SYSTEM MSFUji
  (* Version 1.0, 2021-07-06, HP *)
  APPLICATION MSFFApp
    FBS
      E_CYCLE : E_CYCLE(DT := T#10ms);
      Stage3 : Stage3(DT := 0.01);
      Stage4 : Stage4(DT := 0.01);
      Stage5 : Stage5(DT := 0.01);
      Stage6 : Stage6(DT := 0.01);
      Stage7 : Stage7(DT := 0.01);
      Stage8 : Stage8(DT := 0.01);
      Stage9 : Stage9(DT := 0.01);
      Stage10 : Stage10(DT := 0.01);
      Stage11 : Stage11(DT := 0.01);
      Stage12 : Stage12(DT := 0.01);
      Stage13 : Stage13(DT := 0.01);
      Stage14 : Stage14(DT := 0.01);
      Stage15 : Stage15(DT := 0.01);
      Stage16 : Stage16(DT := 0.01);
      Stage17 : Stage17(DT := 0.01);
      Stage18 : Stage18(DT := 0.01);
      Stage19 : Stage19(DT := 0.01);
      Stage20 : Stage20(WFset := 143.81, DT := 0.01);
      Stage21 : Stage21(DT := 0.01);
      Stagesss22 : Stagesss22(DT := 0.01);
      Stage1 : Stage1(DT := 0.01);
      Stage2 : Stage2(DT := 0.01);
      Stage0 : Stage0(B0set := 217.35, WSset := 2.435, TFEEDset := 35, TSset := 98, DT := 0.01);
    END_FBS
    EVENT_CONNECTIONS
      Stage4.INITO TO Stage5.INIT;
      Stage4.CNF TO Stage5.REQ;
      Stage5.INITO TO Stage6.INIT;
      Stage5.CNF TO Stage6.REQ;
      Stage6.INITO TO Stage7.INIT;
      Stage6.CNF TO Stage7.REQ;
      Stage7.INITO TO Stage8.INIT;
      Stage7.CNF TO Stage8.REQ;
      Stage8.INITO TO Stage9.INIT;
      Stage8.CNF TO Stage9.REQ;
      Stage9.INITO TO Stage10.INIT;
      Stage9.CNF TO Stage10.REQ;
      Stage10.INITO TO Stage11.INIT;
      Stage10.CNF TO Stage11.REQ;
      Stage11.INITO TO Stage12.INIT;
      Stage11.CNF TO Stage12.REQ;
      Stage12.INITO TO Stage13.INIT;
      Stage12.CNF TO Stage13.REQ;
      Stage13.INITO TO Stage14.INIT;
      Stage13.CNF TO Stage14.REQ;
      Stage14.INITO TO Stage15.INIT;
      Stage14.CNF TO Stage15.REQ;
      Stage15.INITO TO Stage16.INIT;
      Stage15.CNF TO Stage16.REQ;
      Stage16.INITO TO Stage17.INIT;
      Stage16.CNF TO Stage17.REQ;
      Stage17.INITO TO Stage18.INIT;
      Stage17.CNF TO Stage18.REQ;
      Stage18.INITO TO Stage19.INIT;
      Stage18.CNF TO Stage19.REQ;
      Stage19.INITO TO Stage20.INIT;
      Stage19.CNF TO Stage20.REQ;
      Stage20.INITO TO Stage21.INIT;
      Stage20.CNF TO Stage21.REQ;
      Stage21.INITO TO Stagesss22.INIT;
      Stage21.CNF TO Stagesss22.REQ;
      Stage3.INITO TO Stage4.INIT;
      Stage3.CNF TO Stage4.REQ;
      Stage1.INITO TO Stage2.INIT;
      Stage1.CNF TO Stage2.REQ;
      E_CYCLE.EO TO Stage0.REQ;
      Stage0.INITO TO Stage1.INIT;
      Stage0.CNF TO Stage1.REQ;
      Stage2.INITO TO Stage3.INIT;
      Stage2.CNF TO Stage3.REQ;
    END_CONNECTIONS
    DATA_CONNECTIONS
      Stage3.B0set TO Stage4.B0set;
      Stage3.WSset TO Stage4.WSset;
      Stage3.TFEEDset TO Stage4.TFEEDset;
      Stage3.DL3 TO Stage4.DL3;
      Stage3.PP3 TO Stage4.PP3;
      Stage3.BR3 TO Stage4.BR3;
      Stage3.TB3 TO Stage4.TB3;
      Stage4.TF4 TO Stage3.TF4;
      Stage4.B0 TO Stage5.B0;
      Stage4.WS TO Stage5.WS;
      Stage4.TFEED TO Stage5.TFEED;
      Stage4.DL4 TO Stage5.DL4;
      Stage4.PP4 TO Stage5.PP4;
      Stage4.BR4 TO Stage5.BR4;
      Stage4.TB4 TO Stage5.TB4;
      Stage5.TF5 TO Stage4.TF5;
      Stage5.B0set TO Stage6.B0set;
      Stage5.WSset TO Stage6.WSset;
      Stage5.TFEEDset TO Stage6.TFEEDset;
      Stage5.DL5 TO Stage6.DL5;
      Stage5.PP5 TO Stage6.PP5;
      Stage5.BR5 TO Stage6.BR5;
      Stage5.TB5 TO Stage6.TB5;
      Stage6.TF6 TO Stage5.TF6;
      Stage6.B0 TO Stage7.B0;
      Stage6.WS TO Stage7.WS;
      Stage6.TFEED TO Stage7.TFEED;
      Stage6.DL6 TO Stage7.DL6;
      Stage6.PP6 TO Stage7.PP6;
      Stage6.BR6 TO Stage7.BR6;
      Stage6.TB6 TO Stage7.TB6;
      Stage7.TF7 TO Stage6.TF7;
      Stage7.B0set TO Stage8.B0set;
      Stage7.WSset TO Stage8.WSset;
      Stage7.TFEEDset TO Stage8.TFEEDset;
      Stage7.DL7 TO Stage8.DL7;
      Stage7.PP7 TO Stage8.PP7;
      Stage7.BR7 TO Stage8.BR7;
      Stage7.TB7 TO Stage8.TB7;
      Stage8.TF8 TO Stage7.TF8;
      Stage8.B0 TO Stage9.B0;
      Stage8.WS TO Stage9.WS;
      Stage8.TFEED TO Stage9.TFEED;
      Stage8.DL8 TO Stage9.DL8;
      Stage8.PP8 TO Stage9.PP8;
      Stage8.BR8 TO Stage9.BR8;
      Stage8.TB8 TO Stage9.TB8;
      Stage9.TF9 TO Stage8.TF9;
      Stage9.B0set TO Stage10.B0set;
      Stage9.WSset TO Stage10.WSset;
      Stage9.TFEEDset TO Stage10.TFEEDset;
      Stage9.DL9 TO Stage10.DL9;
      Stage9.PP9 TO Stage10.PP9;
      Stage9.BR9 TO Stage10.BR9;
      Stage9.TB9 TO Stage10.TB9;
      Stage10.TF10 TO Stage9.TF10;
      Stage10.B0 TO Stage11.B0;
      Stage10.WS TO Stage11.WS;
      Stage10.TFEED TO Stage11.TFEED;
      Stage10.DL10 TO Stage11.DL10;
      Stage10.PP10 TO Stage11.PP10;
      Stage10.BR10 TO Stage11.BR10;
      Stage10.TB10 TO Stage11.TB10;
      Stage11.TF11 TO Stage10.TF11;
      Stage11.B0set TO Stage12.B0set;
      Stage11.WSset TO Stage12.WSset;
      Stage11.TFEEDset TO Stage12.TFEEDset;
      Stage11.DL11 TO Stage12.DL11;
      Stage11.PP11 TO Stage12.PP11;
      Stage11.BR11 TO Stage12.BR11;
      Stage11.TB11 TO Stage12.TB11;
      Stage12.TF12 TO Stage11.TF12;
      Stage12.B0 TO Stage13.B0;
      Stage12.WS TO Stage13.WS;
      Stage12.TFEED TO Stage13.TFEED;
      Stage12.DL12 TO Stage13.DL12;
      Stage12.PP12 TO Stage13.PP12;
      Stage12.BR12 TO Stage13.BR12;
      Stage12.TB12 TO Stage13.TB12;
      Stage13.TF13 TO Stage12.TF13;
      Stage13.B0set TO Stage14.B0set;
      Stage13.WSset TO Stage14.WSset;
      Stage13.TFEEDset TO Stage14.TFEEDset;
      Stage13.DL13 TO Stage14.DL13;
      Stage13.PP13 TO Stage14.PP13;
      Stage13.BR13 TO Stage14.BR13;
      Stage13.TB13 TO Stage14.TB13;
      Stage14.TF14 TO Stage13.TF14;
      Stage14.B0 TO Stage15.B0;
      Stage14.WS TO Stage15.WS;
      Stage14.TFEED TO Stage15.TFEED;
      Stage14.DL14 TO Stage15.DL14;
      Stage14.PP14 TO Stage15.PP14;
      Stage14.BR14 TO Stage15.BR14;
      Stage14.TB14 TO Stage15.TB14;
      Stage15.TF15 TO Stage14.TF15;
      Stage15.B0set TO Stage16.B0set;
      Stage15.WSset TO Stage16.WSset;
      Stage15.TFEEDset TO Stage16.TFEEDset;
      Stage15.DL15 TO Stage16.DL15;
      Stage15.PP15 TO Stage16.PP15;
      Stage15.BR15 TO Stage16.BR15;
      Stage15.TB15 TO Stage16.TB15;
      Stage16.TF16 TO Stage15.TF16;
      Stage16.B0 TO Stage17.B0;
      Stage16.WS TO Stage17.WS;
      Stage16.TFEED TO Stage17.TFEED;
      Stage16.DL16 TO Stage17.DL16;
      Stage16.PP16 TO Stage17.PP16;
      Stage16.BR16 TO Stage17.BR16;
      Stage16.TB16 TO Stage17.TB16;
      Stage17.TF17 TO Stage16.TF17;
      Stage17.B0set TO Stage18.B0set;
      Stage17.WSset TO Stage18.WSset;
      Stage17.TFEEDset TO Stage18.TFEEDset;
      Stage17.DL17 TO Stage18.DL17;
      Stage17.PP17 TO Stage18.PP17;
      Stage17.BR17 TO Stage18.BR17;
      Stage17.TB17 TO Stage18.TB17;
      Stage18.TF18 TO Stage17.TF18;
      Stage18.B0 TO Stage19.B0;
      Stage18.WS TO Stage19.WS;
      Stage18.TFEED TO Stage19.TFEED;
      Stage18.DL18 TO Stage19.DL18;
      Stage18.PP18 TO Stage19.PP18;
      Stage18.BR18 TO Stage19.BR18;
      Stage18.TB18 TO Stage19.TB18;
      Stage19.TF19 TO Stage18.TF19;
      Stage19.B0set TO Stage20.B0set;
      Stage19.WSset TO Stage20.WSset;
      Stage19.TFEEDset TO Stage20.TFEEDset;
      Stage19.DL19 TO Stage20.DL19;
      Stage19.PP19 TO Stage20.PP19;
      Stage19.BR19 TO Stage20.BR19;
      Stage19.TB19 TO Stage20.TB19;
      Stage20.B0 TO Stage21.B0;
      Stage20.WF TO Stage21.WF;
      Stage20.WS TO Stage21.WS;
      Stage20.TFEED TO Stage21.TFEED;
      Stage20.DL20 TO Stage21.DL20;
      Stage20.PP20 TO Stage21.PP20;
      Stage20.BR20 TO Stage21.BR20;
      Stage20.TB20 TO Stage21.TB20;
      Stage21.TF21 TO Stage20.TF21;
      Stage21.B0set TO Stagesss22.B0set;
      Stage21.WFset TO Stagesss22.WFset;
      Stage21.WSset TO Stagesss22.WSset;
      Stage21.TFEEDset TO Stagesss22.TFEEDset;
      Stage21.PP21 TO Stagesss22.PP21;
      Stage21.BR21 TO Stagesss22.BR21;
      Stage21.DL21 TO Stagesss22.DL21;
      Stage21.TB21 TO Stagesss22.TB21;
      Stage20.TF20 TO Stagesss22.TF20;
      Stagesss22.TF22 TO Stage21.TF22;
      Stagesss22.TB22 TO Stage19.TB22;
      Stage1.B0set TO Stage2.B0set;
      Stage1.WSset TO Stage2.WSset;
      Stage1.TFEEDset TO Stage2.TFEEDset;
      Stage1.DL1 TO Stage2.DL1;
      Stage1.PP1 TO Stage2.PP1;
      Stage1.BR1 TO Stage2.BR1;
      Stage1.TB1 TO Stage2.TB1;
      Stage2.TF2 TO Stage1.TF2;
      Stage1.TF1 TO Stage0.TF1;
      Stage0.B0 TO Stage1.B0;
      Stage0.WS TO Stage1.WS;
      Stage0.TFEED TO Stage1.TFEED;
      Stage0.PP0 TO Stage1.PP0;
      Stage0.TB0 TO Stage1.TB0;
      Stage2.B0 TO Stage3.B0;
      Stage2.WS TO Stage3.WS;
      Stage2.TFEED TO Stage3.TFEED;
      Stage2.PP2 TO Stage3.PP2;
      Stage2.BR2 TO Stage3.BR2;
      Stage2.DL2 TO Stage3.DL2;
      Stage2.TB2 TO Stage3.TB2;
      Stage3.TF3 TO Stage2.TF3;
    END_CONNECTIONS
  END_APPLICATION
  DEVICE FORTE_PC : FORTE_PC(MGR_ID := "localhost:61499")
    {SET_ATTRIBUTE(Profile, HOLOBLOC)} (* device profile *)
    RESOURCE MSF : EMB_RES
      FBS
        E_CYCLE : E_CYCLE(DT := T#10ms);
         : Stage0;
         : Stage2;
        Stage3 : Stage3(DT := 0.01);
        Stage4 : Stage4(DT := 0.01);
        Stage5 : Stage5(DT := 0.01);
        Stage6 : Stage6(DT := 0.01);
        Stage7 : Stage7(DT := 0.01);
        Stage8 : Stage8(DT := 0.01);
        Stage9 : Stage9(DT := 0.01);
        Stage10 : Stage10(DT := 0.01);
        Stage11 : Stage11(DT := 0.01);
        Stage12 : Stage12(DT := 0.01);
        Stage13 : Stage13(DT := 0.01);
        Stage14 : Stage14(DT := 0.01);
        Stage15 : Stage15(DT := 0.01);
        Stage16 : Stage16(DT := 0.01);
        Stage17 : Stage17(DT := 0.01);
        Stage18 : Stage18(DT := 0.01);
        Stage19 : Stage19(DT := 0.01);
        Stage20 : Stage20(WFset := 143.81, DT := 0.01);
        Stage21 : Stage21(DT := 0.01);
        Stagesss22 : Stagesss22(DT := 0.01);
        Stage1 : Stage1(DT := 0.01);
        Stage2 : Stage2(DT := 0.01);
        Stage0 : Stage0(B0set := 217.35, WSset := 2.435, TFEEDset := 35, TSset := 98, DT := 0.01);
      END_FBS
      EVENT_CONNECTIONS
        START.COLD TO E_CYCLE.START;
        START.WARM TO E_CYCLE.START;
        Stage4.INITO TO Stage5.INIT;
        Stage4.CNF TO Stage5.REQ;
        Stage5.INITO TO Stage6.INIT;
        Stage5.CNF TO Stage6.REQ;
        Stage6.INITO TO Stage7.INIT;
        Stage6.CNF TO Stage7.REQ;
        Stage7.INITO TO Stage8.INIT;
        Stage7.CNF TO Stage8.REQ;
        Stage8.INITO TO Stage9.INIT;
        Stage8.CNF TO Stage9.REQ;
        Stage9.INITO TO Stage10.INIT;
        Stage9.CNF TO Stage10.REQ;
        Stage10.INITO TO Stage11.INIT;
        Stage10.CNF TO Stage11.REQ;
        Stage11.INITO TO Stage12.INIT;
        Stage11.CNF TO Stage12.REQ;
        Stage12.INITO TO Stage13.INIT;
        Stage12.CNF TO Stage13.REQ;
        Stage13.INITO TO Stage14.INIT;
        Stage13.CNF TO Stage14.REQ;
        Stage14.INITO TO Stage15.INIT;
        Stage14.CNF TO Stage15.REQ;
        Stage15.INITO TO Stage16.INIT;
        Stage15.CNF TO Stage16.REQ;
        Stage16.INITO TO Stage17.INIT;
        Stage16.CNF TO Stage17.REQ;
        Stage17.INITO TO Stage18.INIT;
        Stage17.CNF TO Stage18.REQ;
        Stage18.INITO TO Stage19.INIT;
        Stage18.CNF TO Stage19.REQ;
        Stage19.INITO TO Stage20.INIT;
        Stage19.CNF TO Stage20.REQ;
        Stage20.INITO TO Stage21.INIT;
        Stage20.CNF TO Stage21.REQ;
        Stage21.INITO TO Stagesss22.INIT;
        Stage21.CNF TO Stagesss22.REQ;
        Stage3.INITO TO Stage4.INIT;
        Stage3.CNF TO Stage4.REQ;
        Stage1.INITO TO Stage2.INIT;
        Stage1.CNF TO Stage2.REQ;
        E_CYCLE.EO TO Stage0.REQ;
        Stage0.INITO TO Stage1.INIT;
        Stage0.CNF TO Stage1.REQ;
        START.COLD TO Stage0.INIT;
        START.WARM TO Stage0.INIT;
        Stage2.INITO TO Stage3.INIT;
        Stage2.CNF TO Stage3.REQ;
      END_CONNECTIONS
      DATA_CONNECTIONS
        Stage3.B0set TO Stage4.B0set;
        Stage3.WSset TO Stage4.WSset;
        Stage3.TFEEDset TO Stage4.TFEEDset;
        Stage3.DL3 TO Stage4.DL3;
        Stage3.PP3 TO Stage4.PP3;
        Stage3.BR3 TO Stage4.BR3;
        Stage3.TB3 TO Stage4.TB3;
        Stage4.TF4 TO Stage3.TF4;
        Stage4.B0 TO Stage5.B0;
        Stage4.WS TO Stage5.WS;
        Stage4.TFEED TO Stage5.TFEED;
        Stage4.DL4 TO Stage5.DL4;
        Stage4.PP4 TO Stage5.PP4;
        Stage4.BR4 TO Stage5.BR4;
        Stage4.TB4 TO Stage5.TB4;
        Stage5.TF5 TO Stage4.TF5;
        Stage5.B0set TO Stage6.B0set;
        Stage5.WSset TO Stage6.WSset;
        Stage5.TFEEDset TO Stage6.TFEEDset;
        Stage5.DL5 TO Stage6.DL5;
        Stage5.PP5 TO Stage6.PP5;
        Stage5.BR5 TO Stage6.BR5;
        Stage5.TB5 TO Stage6.TB5;
        Stage6.TF6 TO Stage5.TF6;
        Stage6.B0 TO Stage7.B0;
        Stage6.WS TO Stage7.WS;
        Stage6.TFEED TO Stage7.TFEED;
        Stage6.DL6 TO Stage7.DL6;
        Stage6.PP6 TO Stage7.PP6;
        Stage6.BR6 TO Stage7.BR6;
        Stage6.TB6 TO Stage7.TB6;
        Stage7.TF7 TO Stage6.TF7;
        Stage7.B0set TO Stage8.B0set;
        Stage7.WSset TO Stage8.WSset;
        Stage7.TFEEDset TO Stage8.TFEEDset;
        Stage7.DL7 TO Stage8.DL7;
        Stage7.PP7 TO Stage8.PP7;
        Stage7.BR7 TO Stage8.BR7;
        Stage7.TB7 TO Stage8.TB7;
        Stage8.TF8 TO Stage7.TF8;
        Stage8.B0 TO Stage9.B0;
        Stage8.WS TO Stage9.WS;
        Stage8.TFEED TO Stage9.TFEED;
        Stage8.DL8 TO Stage9.DL8;
        Stage8.PP8 TO Stage9.PP8;
        Stage8.BR8 TO Stage9.BR8;
        Stage8.TB8 TO Stage9.TB8;
        Stage9.TF9 TO Stage8.TF9;
        Stage9.B0set TO Stage10.B0set;
        Stage9.WSset TO Stage10.WSset;
        Stage9.TFEEDset TO Stage10.TFEEDset;
        Stage9.DL9 TO Stage10.DL9;
        Stage9.PP9 TO Stage10.PP9;
        Stage9.BR9 TO Stage10.BR9;
        Stage9.TB9 TO Stage10.TB9;
        Stage10.TF10 TO Stage9.TF10;
        Stage10.B0 TO Stage11.B0;
        Stage10.WS TO Stage11.WS;
        Stage10.TFEED TO Stage11.TFEED;
        Stage10.DL10 TO Stage11.DL10;
        Stage10.PP10 TO Stage11.PP10;
        Stage10.BR10 TO Stage11.BR10;
        Stage10.TB10 TO Stage11.TB10;
        Stage11.TF11 TO Stage10.TF11;
        Stage11.B0set TO Stage12.B0set;
        Stage11.WSset TO Stage12.WSset;
        Stage11.TFEEDset TO Stage12.TFEEDset;
        Stage11.DL11 TO Stage12.DL11;
        Stage11.PP11 TO Stage12.PP11;
        Stage11.BR11 TO Stage12.BR11;
        Stage11.TB11 TO Stage12.TB11;
        Stage12.TF12 TO Stage11.TF12;
        Stage12.B0 TO Stage13.B0;
        Stage12.WS TO Stage13.WS;
        Stage12.TFEED TO Stage13.TFEED;
        Stage12.DL12 TO Stage13.DL12;
        Stage12.PP12 TO Stage13.PP12;
        Stage12.BR12 TO Stage13.BR12;
        Stage12.TB12 TO Stage13.TB12;
        Stage13.TF13 TO Stage12.TF13;
        Stage13.B0set TO Stage14.B0set;
        Stage13.WSset TO Stage14.WSset;
        Stage13.TFEEDset TO Stage14.TFEEDset;
        Stage13.DL13 TO Stage14.DL13;
        Stage13.PP13 TO Stage14.PP13;
        Stage13.BR13 TO Stage14.BR13;
        Stage13.TB13 TO Stage14.TB13;
        Stage14.TF14 TO Stage13.TF14;
        Stage14.B0 TO Stage15.B0;
        Stage14.WS TO Stage15.WS;
        Stage14.TFEED TO Stage15.TFEED;
        Stage14.DL14 TO Stage15.DL14;
        Stage14.PP14 TO Stage15.PP14;
        Stage14.BR14 TO Stage15.BR14;
        Stage14.TB14 TO Stage15.TB14;
        Stage15.TF15 TO Stage14.TF15;
        Stage15.B0set TO Stage16.B0set;
        Stage15.WSset TO Stage16.WSset;
        Stage15.TFEEDset TO Stage16.TFEEDset;
        Stage15.DL15 TO Stage16.DL15;
        Stage15.PP15 TO Stage16.PP15;
        Stage15.BR15 TO Stage16.BR15;
        Stage15.TB15 TO Stage16.TB15;
        Stage16.TF16 TO Stage15.TF16;
        Stage16.B0 TO Stage17.B0;
        Stage16.WS TO Stage17.WS;
        Stage16.TFEED TO Stage17.TFEED;
        Stage16.DL16 TO Stage17.DL16;
        Stage16.PP16 TO Stage17.PP16;
        Stage16.BR16 TO Stage17.BR16;
        Stage16.TB16 TO Stage17.TB16;
        Stage17.TF17 TO Stage16.TF17;
        Stage17.B0set TO Stage18.B0set;
        Stage17.WSset TO Stage18.WSset;
        Stage17.TFEEDset TO Stage18.TFEEDset;
        Stage17.DL17 TO Stage18.DL17;
        Stage17.PP17 TO Stage18.PP17;
        Stage17.BR17 TO Stage18.BR17;
        Stage17.TB17 TO Stage18.TB17;
        Stage18.TF18 TO Stage17.TF18;
        Stage18.B0 TO Stage19.B0;
        Stage18.WS TO Stage19.WS;
        Stage18.TFEED TO Stage19.TFEED;
        Stage18.DL18 TO Stage19.DL18;
        Stage18.PP18 TO Stage19.PP18;
        Stage18.BR18 TO Stage19.BR18;
        Stage18.TB18 TO Stage19.TB18;
        Stage19.TF19 TO Stage18.TF19;
        Stage19.B0set TO Stage20.B0set;
        Stage19.WSset TO Stage20.WSset;
        Stage19.TFEEDset TO Stage20.TFEEDset;
        Stage19.DL19 TO Stage20.DL19;
        Stage19.PP19 TO Stage20.PP19;
        Stage19.BR19 TO Stage20.BR19;
        Stage19.TB19 TO Stage20.TB19;
        Stage20.B0 TO Stage21.B0;
        Stage20.WF TO Stage21.WF;
        Stage20.WS TO Stage21.WS;
        Stage20.TFEED TO Stage21.TFEED;
        Stage20.DL20 TO Stage21.DL20;
        Stage20.PP20 TO Stage21.PP20;
        Stage20.BR20 TO Stage21.BR20;
        Stage20.TB20 TO Stage21.TB20;
        Stage21.TF21 TO Stage20.TF21;
        Stage21.B0set TO Stagesss22.B0set;
        Stage21.WFset TO Stagesss22.WFset;
        Stage21.WSset TO Stagesss22.WSset;
        Stage21.TFEEDset TO Stagesss22.TFEEDset;
        Stage21.DL21 TO Stagesss22.DL21;
        Stage21.PP21 TO Stagesss22.PP21;
        Stage21.BR21 TO Stagesss22.BR21;
        Stage21.TB21 TO Stagesss22.TB21;
        Stage20.TF20 TO Stagesss22.TF20;
        Stagesss22.TF22 TO Stage21.TF22;
        Stagesss22.TB22 TO Stage19.TB22;
        Stage1.B0set TO Stage2.B0set;
        Stage1.WSset TO Stage2.WSset;
        Stage1.TFEEDset TO Stage2.TFEEDset;
        Stage1.DL1 TO Stage2.DL1;
        Stage1.PP1 TO Stage2.PP1;
        Stage1.BR1 TO Stage2.BR1;
        Stage1.TB1 TO Stage2.TB1;
        Stage2.TF2 TO Stage1.TF2;
        Stage1.TF1 TO Stage0.TF1;
        Stage0.B0 TO Stage1.B0;
        Stage0.WS TO Stage1.WS;
        Stage0.TFEED TO Stage1.TFEED;
        Stage0.PP0 TO Stage1.PP0;
        Stage0.TB0 TO Stage1.TB0;
        Stage2.B0 TO Stage3.B0;
        Stage2.WS TO Stage3.WS;
        Stage2.TFEED TO Stage3.TFEED;
        Stage2.PP2 TO Stage3.PP2;
        Stage2.BR2 TO Stage3.BR2;
        Stage2.DL2 TO Stage3.DL2;
        Stage2.TB2 TO Stage3.TB2;
        Stage3.TF3 TO Stage2.TF3;
      END_CONNECTIONS
    END_RESOURCE
  END_DEVICE
  MAPPINGS
    MSFFApp.E_CYCLE ON FORTE_PC.MSF.E_CYCLE;
    MSFFApp.Stage3 ON FORTE_PC.MSF.Stage3;
    MSFFApp.Stage4 ON FORTE_PC.MSF.Stage4;
    MSFFApp.Stage5 ON FORTE_PC.MSF.Stage5;
    MSFFApp.Stage6 ON FORTE_PC.MSF.Stage6;
    MSFFApp.Stage7 ON FORTE_PC.MSF.Stage7;
    MSFFApp.Stage8 ON FORTE_PC.MSF.Stage8;
    MSFFApp.Stage9 ON FORTE_PC.MSF.Stage9;
    MSFFApp.Stage10 ON FORTE_PC.MSF.Stage10;
    MSFFApp.Stage11 ON FORTE_PC.MSF.Stage11;
    MSFFApp.Stage12 ON FORTE_PC.MSF.Stage12;
    MSFFApp.Stage13 ON FORTE_PC.MSF.Stage13;
    MSFFApp.Stage14 ON FORTE_PC.MSF.Stage14;
    MSFFApp.Stage15 ON FORTE_PC.MSF.Stage15;
    MSFFApp.Stage16 ON FORTE_PC.MSF.Stage16;
    MSFFApp.Stage17 ON FORTE_PC.MSF.Stage17;
    MSFFApp.Stage18 ON FORTE_PC.MSF.Stage18;
    MSFFApp.Stage19 ON FORTE_PC.MSF.Stage19;
    MSFFApp.Stage20 ON FORTE_PC.MSF.Stage20;
    MSFFApp.Stage21 ON FORTE_PC.MSF.Stage21;
    MSFFApp.Stagesss22 ON FORTE_PC.MSF.Stagesss22;
    MSFFApp.Stage1 ON FORTE_PC.MSF.Stage1;
    MSFFApp.Stage2 ON FORTE_PC.MSF.Stage2;
    MSFFApp.Stage0 ON FORTE_PC.MSF.Stage0;
  END_MAPPINGS
  SEGMENTS
    Ethernet : Ethernet;
  END_SEGMENTS
  LINKS
    FORTE_PC => Ethernet;
  END_LINKS
END_SYSTEM
